PROGRAM main
VAR
	Enable AT %QX0.0 : bool;
	DelayTimer : TON;
	Output AT %QX0.1 : bool;
	TimerElapsed : time;
	ElapsedSeconds AT %MD0 : dint;
END_VAR

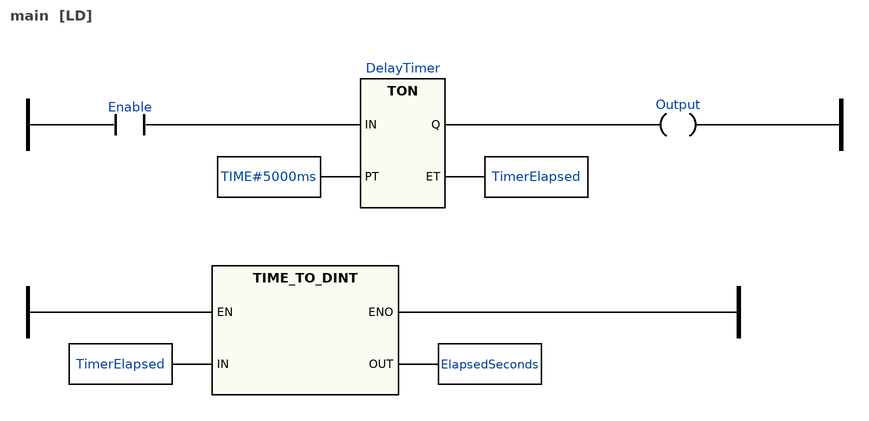
(* LD diagram, written out as Structured Text *)
DelayTimer(IN := Enable, PT := TIME#5000ms);
Output := DelayTimer.Q;
TimerElapsed := DelayTimer.ET;
ElapsedSeconds := TIME_TO_DINT(TimerElapsed);
END_PROGRAM
